// TIA Portal V21 export
DATA_BLOCK "DATALOG"   // DB309
{ S7_Optimized_Access := 'FALSE' }
   VAR RETAIN
      "SET PRINT INTERVAL" : Int;
      "PROCESS PHASE" : Int;
      "TRIGGER BIT" : Bool;
      "START/STOP" : Bool;
      "BATCH DATA" : Struct
         "BATCH CODE" : WString;
         "BATCH NAME" : WString;
         "EQUIPMENT ID" : WString;
         "OPERATOR NAME" : WString;
         "PRODUCT NAME" : WString;
         "START DATE STRING" : WString;
         "END DATE STRING" : WString;
      END_STRUCT;
      INTERLOCK : Struct
         VACCUM : Struct
            START : Bool;
            STOP : Bool;
            NEW : Bool;
            BUFF : Int;
         END_STRUCT;
      END_STRUCT;
   END_VAR
BEGIN
END_DATA_BLOCK
